// TIA Portal V19 export
TYPE "C215_VAR_SVLU_TYPIC"
   STRUCT
      STS { ExternalAccessible := 'False'; ExternalVisible := 'False'; ExternalWritable := 'False'} : USInt;   // Status van het statisch indicatiebord vluchtroute
      BST { ExternalAccessible := 'False'; ExternalVisible := 'False'; ExternalWritable := 'False'} : USInt;   // Bestuurbaarheid
   END_STRUCT;
END_TYPE
